# EPICS autosave request: support/optics/2-6-1/opticsApp/Db/Io_settings.req
$(P)scaler
$(P)xAir
$(P)xN2
$(P)xHe
$(P)xAr
$(P)xCO2
$(P)v2f
$(P)VperA
$(P)HePath
$(P)airPath
$(P)Be
$(P)efficiency
$(P)ArPcntr
$(P)activeLen
$(P)deadFront
$(P)deadRear
$(P)kapton1
$(P)kapton2
